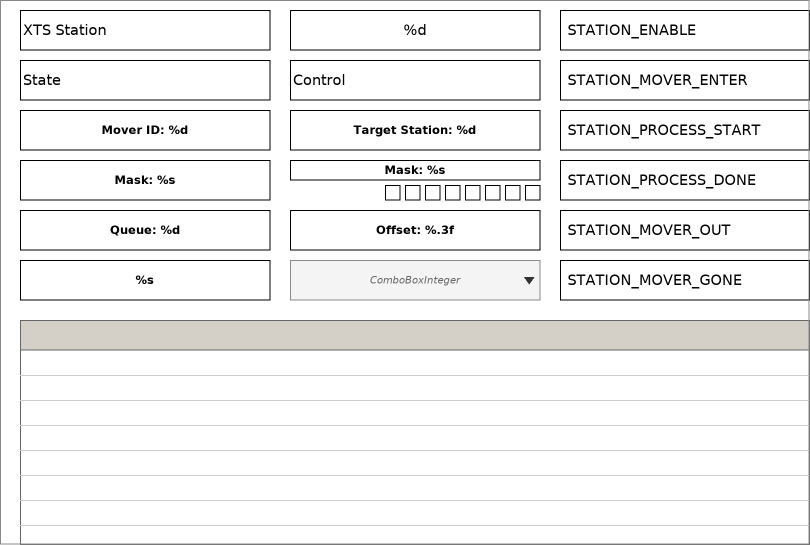
VISUALIZATION STATION_VISU  // 810x545
    Rectangle (20,10 250x40), "XTS Station"
    Rectangle (290,10 250x40), "%d", text variable: MAIN.nStationSelected
        OnMouseClick: write the text variable via VisuDialogs.Numpad, min 1, max MAX_STATION, title 'Selected Station'
    Rectangle (20,60 250x40), "State"
    Rectangle (290,60 250x40), "Control"
    Rectangle (20,210 250x40), "Queue: %d", text variable: GVL_XTS.StationState[MAIN.nStationSelected].nQueue
    Rectangle (20,110 250x40), "Mover ID: %d", text variable: GVL_XTS.StationState[MAIN.nStationSelected].nMoverId
    Rectangle (20,160 250x40), "Mask: %s", text variable: MAIN.sStationStateMask
    Rectangle (20,260 250x40), "%s", text variable: MAIN.sStationState
    ComboBoxInteger (290,260 250x40), variable: GVL_XTS.StationCtrl[MAIN.nStationSelected].eCmd, text list: 'TL_E_CTRL_STATION'
    Rectangle (290,210 250x40), "Offset: %.3f", text variable: GVL_XTS.StationCtrl[MAIN.nStationSelected].rOffset
    Rectangle (290,110 250x40), "Target Station: %d", text variable: GVL_XTS.StationCtrl[MAIN.nStationSelected].nTargetStation
        OnMouseClick: write the text variable via VisuDialogs.Numpad, min 1, max MAX_STATION, title 'Target Station'
    Rectangle (290,160 250x20), "Mask: %s", text variable: MAIN.sStationCtrlMask
    Rectangle (525,185 15x15)
        toggle GVL_XTS.StationCtrl[MAIN.nStationSelected].nMask.0
    Rectangle (505,185 15x15)
        toggle GVL_XTS.StationCtrl[MAIN.nStationSelected].nMask.1
    Rectangle (485,185 15x15)
        toggle GVL_XTS.StationCtrl[MAIN.nStationSelected].nMask.2
    Rectangle (465,185 15x15)
        toggle GVL_XTS.StationCtrl[MAIN.nStationSelected].nMask.3
    Rectangle (445,185 15x15)
        toggle GVL_XTS.StationCtrl[MAIN.nStationSelected].nMask.4
    Rectangle (425,185 15x15)
        toggle GVL_XTS.StationCtrl[MAIN.nStationSelected].nMask.5
    Rectangle (405,185 15x15)
        toggle GVL_XTS.StationCtrl[MAIN.nStationSelected].nMask.6
    Rectangle (385,185 15x15)
        toggle GVL_XTS.StationCtrl[MAIN.nStationSelected].nMask.7
    Rectangle (560,10 250x40), "STATION_ENABLE", colour toggle: MAIN.bStationEnable
        OnMouseClick: execute { GVL_XTS.StationCtrl[MAIN.nStationSelected].eCmd := E_STATION_CTRL.STATION_ENABLE; }
    Rectangle (560,60 250x40), "STATION_MOVER_ENTER", colour toggle: MAIN.bStationEnter
        OnMouseClick: execute { GVL_XTS.StationCtrl[MAIN.nStationSelected].eCmd := E_STATION_CTRL.STATION_MOVER_ENTER; }
    Rectangle (560,110 250x40), "STATION_PROCESS_START", colour toggle: MAIN.bStationStart
        OnMouseClick: execute { GVL_XTS.StationCtrl[MAIN.nStationSelected].eCmd := E_STATION_CTRL.STATION_PROCESS_START; }
    Rectangle (560,160 250x40), "STATION_PROCESS_DONE", colour toggle: MAIN.bStationDone
        OnMouseClick: execute { GVL_XTS.StationCtrl[MAIN.nStationSelected].eCmd := E_STATION_CTRL.STATION_PROCESS_DONE; }
    Rectangle (560,210 250x40), "STATION_MOVER_OUT", colour toggle: MAIN.bStationOut
        OnMouseClick: execute { GVL_XTS.StationCtrl[MAIN.nStationSelected].eCmd := E_STATION_CTRL.STATION_MOVER_OUT; }
    Rectangle (560,260 250x40), "STATION_MOVER_GONE", colour toggle: MAIN.bStationGone
        OnMouseClick: execute { GVL_XTS.StationCtrl[MAIN.nStationSelected].eCmd := E_STATION_CTRL.STATION_MOVER_GONE; }
    Table (20,320 790x225), data array: MAIN.tStationSelectedQueue
        p3854506369: MAIN.tStationSelectedQueue[INDEX].nMoverId
        p1892666644: MAIN.tStationSelectedQueue[INDEX].nTargetStation
        p338671338: MAIN.tStationSelectedQueue[INDEX].nMask
        p2170511999: MAIN.tStationSelectedQueue[INDEX].rOffset
END_VISUALIZATION

(* stored: Version 1.1.0.1
   Visu STATION_VISU: Id {4eb84cda-22b7-4c33-965e-9b07ef0c4d4f} *)
